FUNCTION_BLOCK E_TO_UINT (* Event to UINT converter (1 of 4) *)
  (* Standard: 61499-1; Classification: Event processing; Function: Event to integer compression; Type: UINT *)
  (* Version 0.0, 2003-04-10, JHC, Rockwell Automation *)
  (* Compiler header: package fb.rt.events; *)
  (* Compiler Java IBM Jikes 1.06 *)
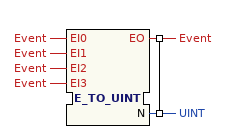
  EVENT_INPUT
    EI0;
    EI1;
    EI2;
    EI3;
  END_EVENT
  EVENT_OUTPUT
    EO WITH N;
  END_EVENT
  VAR_OUTPUT
    N : UINT; (* Event number (0..4) *)
  END_VAR
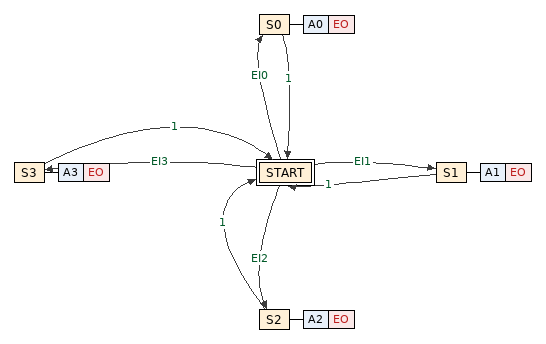
  EC_STATES
    START; (* Initial State *)
    S0 : A0 -> EO;
    S1 : A1 -> EO;
    S2 : A2 -> EO;
    S3 : A3 -> EO;
  END_STATES
  EC_TRANSITIONS
    START TO S0 := EI0;
    START TO S1 := EI1;
    START TO S2 := EI2;
    START TO S3 := EI3;
    S0 TO START := 1;
    S1 TO START := 1;
    S2 TO START := 1;
    S3 TO START := 1;
  END_TRANSITIONS
  ALGORITHM A0 IN ST:
N := 0;
  END_ALGORITHM
  ALGORITHM A1 IN ST:
N := 1;
  END_ALGORITHM
  ALGORITHM A2 IN ST:
N := 2;
  END_ALGORITHM
  ALGORITHM A3 IN ST:
N := 3;
  END_ALGORITHM
END_FUNCTION_BLOCK
